TYPE EtcMasterBase_62654B43 :
STRUCT
END_STRUCT
END_TYPE

(* stored: Version 1.2.0.0, ProductVersion 3.1.4024.9
   DUT EtcMasterBase_62654B43: Id {07f5e1c4-6587-4fe2-a6e5-41faf4aa7c77} *)
